(* PLC project MotionTest1, Higen MCL 1 *)
(* stored: creationDateTime 2012-01-06T15:20:13, modificationDateTime 2013-08-23T10:02:24 *)

FUNCTION_BLOCK PrepAxis
  VAR
    switch : MC_Power;
    readpos : MC_ReadActualPosition;
    readspeed : MC_ReadParameter;
  END_VAR
  VAR_INPUT
    Pwr : BOOL;
  END_VAR
  VAR
    MC_Sim1 : MC_Sim;
  END_VAR
  VAR_OUTPUT
    Axis : AXIS_REF;
    Position : LREAL;
    Velocity : LREAL;
  END_VAR

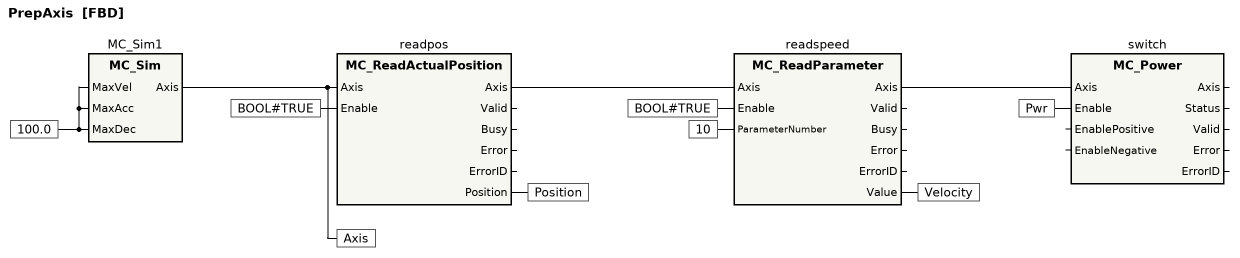
(* FBD diagram, written out as Structured Text *)
MC_Sim1(MaxVel := 100.0, MaxAcc := 100.0, MaxDec := 100.0);
Axis := MC_Sim1.Axis;
readpos(Axis := MC_Sim1.Axis, Enable := BOOL#TRUE);
Position := readpos.Position;
readspeed(Axis := readpos.Axis, Enable := BOOL#TRUE, ParameterNumber := 10);
Velocity := readspeed.Value;
switch(Axis := readspeed.Axis, Enable := Pwr);
END_FUNCTION_BLOCK

FUNCTION_BLOCK wxgetval
  VAR
    getpy : python_gear;
    latch : SR;
  END_VAR
  VAR_INPUT
    name : STRING;
  END_VAR
  VAR_OUTPUT
    val : BOOL;
  END_VAR
  VAR  (* added by the conversion: wires and edge detectors of the diagram *)
    _EQ41_ENO : BOOL;
    _EQ41_OUT : BOOL;
    _EQ3_ENO : BOOL;
    _EQ3_OUT : BOOL;
  END_VAR

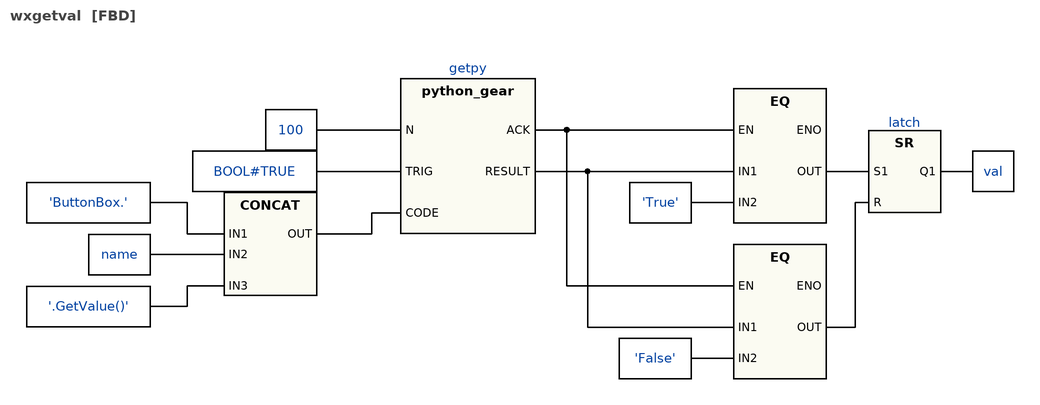
(* FBD diagram, written out as Structured Text *)
getpy(N := 100, TRIG := BOOL#TRUE, CODE := CONCAT('ButtonBox.', name, '.GetValue()'));
_EQ41_OUT := EQ(EN := getpy.ACK, IN1 := getpy.RESULT, IN2 := 'True', ENO => _EQ41_ENO);
_EQ3_OUT := EQ(EN := getpy.ACK, IN1 := getpy.RESULT, IN2 := 'False', ENO => _EQ3_ENO);
latch(S1 := _EQ41_OUT, R := _EQ3_OUT);
val := latch.Q1;
END_FUNCTION_BLOCK

(* - *)
PROGRAM main
  VAR
    AxisX : AXIS_REF;
    AxisY : AXIS_REF;
    AxisZ : AXIS_REF;
    Table : AXIS_REF;
    pX : LREAL;
    pY : LREAL;
    pZ : LREAL;
    vX : LREAL;
    vY : LREAL;
    vZ : LREAL;
    bt1 : wxgetval;
    pb : LREAL;
    vb : LREAL;
    Block1 : wxgetval;
    Block2 : wxgetval;
    Block3 : wxgetval;
    Block6 : wxgetval;
    Block4 : wxgetval;
    Block7 : wxgetval;
    MC_IndexIdentInGroup0 : MC_IndexIdentInGroup;
    MC_AddAxisToGroup0 : MC_AddAxisToGroup;
    MC_CreateAxesGroup0 : MC_CreateAxesGroup;
    MC_AddAxisToGroup1 : MC_AddAxisToGroup;
    MC_IndexIdentInGroup1 : MC_IndexIdentInGroup;
    MC_GroupSetPosition0 : MC_GroupSetPosition;
    MC_ToRealArray0 : MC_ToRealArray;
    MC_GroupEnable0 : MC_GroupEnable;
    MC_AddAxisToGroup2 : MC_AddAxisToGroup;
    MC_IndexIdentInGroup2 : MC_IndexIdentInGroup;
    PrepAxis0 : PrepAxis;
    PrepAxis1 : PrepAxis;
    PrepAxis2 : PrepAxis;
    Group : AXES_GROUP_REF;
    MC_MoveDirectAbsolute0 : MC_MoveDirectAbsolute;
    MC_ToRealArray3 : MC_ToRealArray;
    PrepAxis3 : PrepAxis;
    MC_TrackRotaryTable0 : MC_TrackRotaryTable;
    MC_ToRealArray1 : MC_ToRealArray;
    MC_MoveVelocity0 : MC_MoveVelocity;
    MC_ToRealArray2 : MC_ToRealArray;
    MC_ToRealArray4 : MC_ToRealArray;
    MC_ToRealArray5 : MC_ToRealArray;
    MC_MoveCircularAbsolute1 : MC_MoveCircularAbsolute;
    MC_MoveDirectAbsolute1 : MC_MoveDirectAbsolute;
    MC_ToRealArray6 : MC_ToRealArray;
    MC_SetCartesianTransform0 : MC_SetCartesianTransform;
    MC_ReadCartesianTransform0 : MC_ReadCartesianTransform;
    MC_MoveLinearAbsolute0 : MC_MoveLinearAbsolute;
    MC_ToRealArray7 : MC_ToRealArray;
    MC_ToRealArray8 : MC_ToRealArray;
    MC_MoveLinearRelative0 : MC_MoveLinearRelative;
  END_VAR

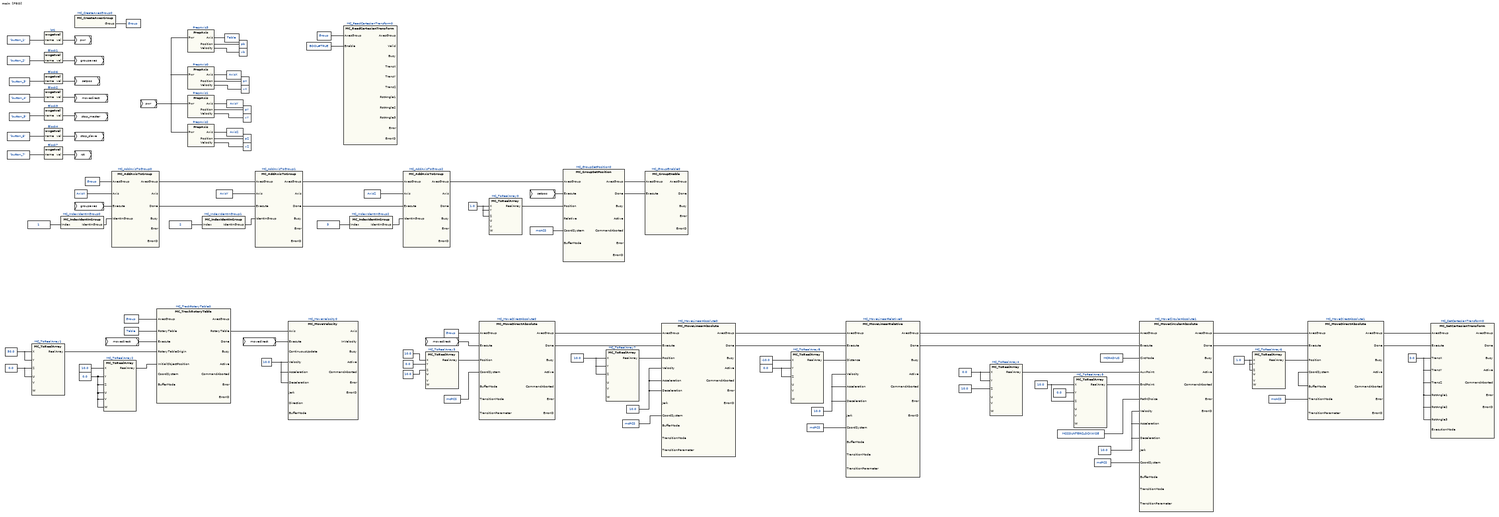
(* FBD diagram, written out as Structured Text *)
MC_CreateAxesGroup0();
Group := MC_CreateAxesGroup0.Group;
bt1(name := 'button_1');
PrepAxis3(Pwr := bt1.val);
Table := PrepAxis3.Axis;
pb := PrepAxis3.Position;
vb := PrepAxis3.Velocity;
PrepAxis0(Pwr := bt1.val);
AxisX := PrepAxis0.Axis;
pX := PrepAxis0.Position;
vX := PrepAxis0.Velocity;
PrepAxis1(Pwr := bt1.val);
AxisY := PrepAxis1.Axis;
pY := PrepAxis1.Position;
vY := PrepAxis1.Velocity;
PrepAxis2(Pwr := bt1.val);
AxisZ := PrepAxis2.Axis;
pZ := PrepAxis2.Position;
vZ := PrepAxis2.Velocity;
MC_ReadCartesianTransform0(AxesGroup := Group, Enable := BOOL#TRUE);
Block1(name := 'button_2');
Block6(name := 'button_3');
Block2(name := 'button_4');
Block3(name := 'button_5');
Block4(name := 'button_6');
Block7(name := 'button_7');
MC_IndexIdentInGroup0(Index := 1);
MC_AddAxisToGroup0(AxesGroup := Group, Axis := AxisX, Execute := Block1.val, IdentInGroup := MC_IndexIdentInGroup0.IdentInGroup);
MC_IndexIdentInGroup1(Index := 2);
MC_AddAxisToGroup1(AxesGroup := MC_AddAxisToGroup0.AxesGroup, Axis := AxisY, Execute := MC_AddAxisToGroup0.Done, IdentInGroup := MC_IndexIdentInGroup1.IdentInGroup);
MC_IndexIdentInGroup2(Index := 3);
MC_AddAxisToGroup2(AxesGroup := MC_AddAxisToGroup1.AxesGroup, Axis := AxisZ, Execute := MC_AddAxisToGroup1.Done, IdentInGroup := MC_IndexIdentInGroup2.IdentInGroup);
MC_ToRealArray0(X := 1.0, Y := 1.0, Z := 1.0);
MC_GroupSetPosition0(AxesGroup := MC_AddAxisToGroup2.AxesGroup, Execute := Block6.val, Position := MC_ToRealArray0.RealArray, CoordSystem := mcACS);
MC_GroupEnable0(AxesGroup := MC_GroupSetPosition0.AxesGroup, Execute := MC_GroupSetPosition0.Done);
MC_ToRealArray1(X := 50.0, Y := 50.0, Z := 0.0, U := 0.0);
MC_ToRealArray2(X := 10.0, Y := 0.0, Z := 0.0, U := 0.0, V := 0.0, W := 0.0);
MC_TrackRotaryTable0(AxesGroup := Group, RotaryTable := Table, Execute := Block2.val, RotaryTableOrigin := MC_ToRealArray1.RealArray, InitialObjectPosition := MC_ToRealArray2.RealArray);
MC_MoveVelocity0(Axis := MC_TrackRotaryTable0.RotaryTable, Execute := Block2.val, Velocity := 10.0, Acceleration := 10.0, Deceleration := 10.0);
MC_ToRealArray3(X := 10.0, Y := 0.0, Z := 10.0);
MC_MoveDirectAbsolute0(AxesGroup := Group, Execute := Block2.val, Position := MC_ToRealArray3.RealArray, CoordSystem := mcPCS);
MC_ToRealArray7(X := 10.0, Y := 10.0, Z := 10.0);
MC_MoveLinearAbsolute0(AxesGroup := MC_MoveDirectAbsolute0.AxesGroup, Execute := MC_MoveDirectAbsolute0.Done, Position := MC_ToRealArray7.RealArray, Velocity := 10.0, Acceleration := 10.0, Deceleration := 10.0, CoordSystem := mcPCS);
MC_ToRealArray8(X := -10.0, Y := 0.0, Z := 0.0);
MC_MoveLinearRelative0(AxesGroup := MC_MoveLinearAbsolute0.AxesGroup, Execute := MC_MoveLinearAbsolute0.Done, Distance := MC_ToRealArray8.RealArray, Velocity := 10.0, Acceleration := 10.0, Deceleration := 10.0, CoordSystem := mcPCS);
MC_ToRealArray4(X := 0.0, Y := 0.0, Z := 10.0);
MC_ToRealArray5(X := 10.0, Y := 0.0, Z := 10.0);
MC_MoveCircularAbsolute1(AxesGroup := MC_MoveLinearRelative0.AxesGroup, Execute := MC_MoveLinearRelative0.Done, CircMode := MCRADIUS, AuxPoint := MC_ToRealArray4.RealArray, EndPoint := MC_ToRealArray5.RealArray, PathChoice := MCCOUNTERCLOCKWISE, Velocity := 10.0, Acceleration := 10.0, Deceleration := 10.0, CoordSystem := mcPCS);
MC_ToRealArray6(X := 1.0, Y := 1.0, Z := 1.0);
MC_MoveDirectAbsolute1(AxesGroup := MC_MoveCircularAbsolute1.AxesGroup, Execute := MC_MoveCircularAbsolute1.Done, Position := MC_ToRealArray6.RealArray, CoordSystem := mcACS);
MC_SetCartesianTransform0(AxesGroup := MC_MoveDirectAbsolute1.AxesGroup, Execute := MC_MoveDirectAbsolute1.Done, TransX := 0.0, TransY := 0.0, TransZ := 0.0, RotAngle1 := 0.0, RotAngle2 := 0.0, RotAngle3 := 0.0);
END_PROGRAM

CONFIGURATION conf
  RESOURCE res ON PLC
    TASK milisecond(INTERVAL := T#10ms, PRIORITY := 0);
    PROGRAM maininstance WITH milisecond : main;
  END_RESOURCE
END_CONFIGURATION
